FUNCTION_BLOCK DataPanel_MI_QW_PWMi (* Output service interface function block for Current Controlled PWM output data (Current Mode 4) *)
  (* Description: Copyright (c) 2026 HR Agrartechnik GmbH *)
  (* Version 1.0, 2026-01-16, generated, HR Agrartechnik GmbH *)
  PACKAGE DataPanel::io::MI::DQ;
  IMPORT DataPanel::io::MI::DQ::DataPanel_MI_DO::Invalid;
  IMPORT DataPanel::io::MI::const::MI;
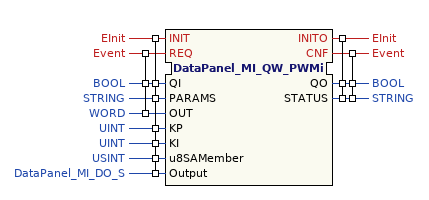
  EVENT_INPUT
    INIT : EInit WITH QI, PARAMS, u8SAMember, Output, KP, KI; (* Service Initialization *)
    REQ WITH QI, OUT; (* Service Request *)
  END_EVENT
  EVENT_OUTPUT
    INITO : EInit WITH QO, STATUS; (* Initialization Confirm *)
    CNF WITH QO, STATUS; (* Confirmation of Requested Service *)
  END_EVENT
  VAR_INPUT
    QI : BOOL; (* Event Input Qualifier *)
    PARAMS : STRING; (* Service Parameters *)
    OUT : WORD; (* Output data to resource *)
    KP : UINT := 70; (* Proportional gain for current control *)
    KI : UINT := 30; (* Integral gain for current control *)
    u8SAMember : USINT := MI::MI_00; (* Node SA 224..239 *)
    Output : DataPanel::io::MI::DQ::DataPanel_MI_DO_S := Invalid; (* Identify the Output DigitalOutput_1A..8B and Input_Power_Port_5..8 *)
  END_VAR
  VAR_OUTPUT
    QO : BOOL; (* Event Output Qualifier *)
    STATUS : STRING; (* Service Status *)
  END_VAR
END_FUNCTION_BLOCK
